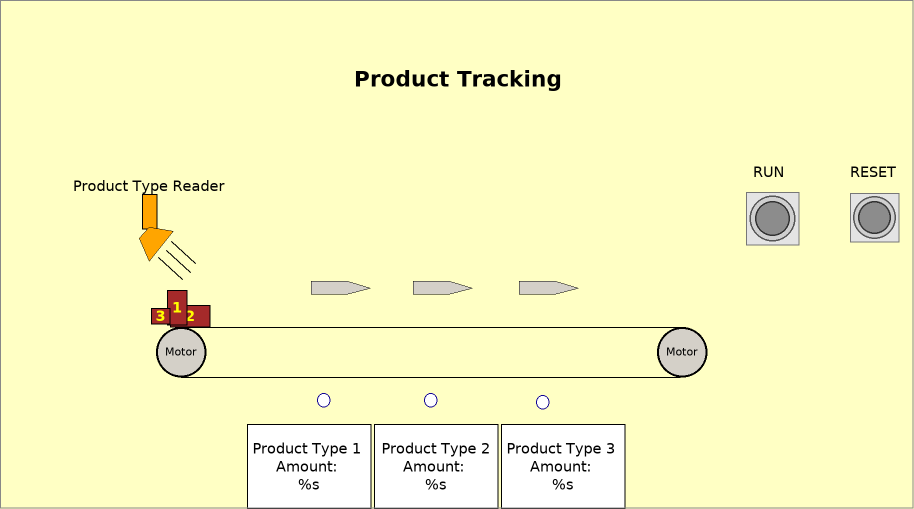
VISUALIZATION Visualization  // 914x509
    PushSwitchLed (746,191 53x55), variable: Simulation.CmdDrv01, behaviour: TOGGLE, style: Switch-PushSwitchLed-Gray
    Ellipse (156,327 50x50), "Motor", colour toggle: Simulation.Drive01.DrvRunning
    Label (728,157 82x30), "RUN"
    Label (832,157 82x30), "RESET"
    Ellipse (657,327 50x50), "Motor", colour toggle: Simulation.Drive01.DrvRunning
    Line (183,327) (680,327)
    Rectangle (142,194 15x35), angle 310
    Label (64,171 170x30), "Product Type Reader"
    Line (181,377) (680,377)
    Polygon (311,281) (347,281) (370,288) (347,294) (311,294)
        p2858320360: BOOL_TO_INT(MAIN.ConveyorTracking01.DiverterCmd) * 90
    Polygon (413,281) (449,281) (472,288) (449,294) (413,294)
        p2858320360: BOOL_TO_INT(MAIN.ConveyorTracking02.DiverterCmd) * 90
    Polygon (519,281) (555,281) (578,288) (555,294) (519,294)
        p2858320360: BOOL_TO_INT(MAIN.ConveyorTracking03.DiverterCmd) * 90
    Rectangle (170,305 40x22), "2", invisible if: Simulation.ProductType <> 2 OR MAIN.ConveyorTracking02.DistanceMoved > 52
        p3560616238: MAIN.ConveyorTracking02.DistanceMoved * 3.9
    Rectangle (167,290 20x35), "1", invisible if: Simulation.ProductType <> 1 OR MAIN.ConveyorTracking01.DistanceMoved > 32
        p3560616238: MAIN.ConveyorTracking01.DistanceMoved * 4.0
    Rectangle (151,308 19x16), "3", invisible if: Simulation.ProductType <> 3 OR MAIN.ConveyorTracking03.DistanceMoved > 72
        p3560616238: MAIN.ConveyorTracking03.DistanceMoved * 4.8
    Rectangle (247,424 124x85), "Product Type 1 Amount: %s", text variable: MAIN.DroppedProducts1.CV
    Ellipse (317,393 13x14), colour toggle: Simulation.tonProdType1Dropped.Q
    Ellipse (424,393 13x14), colour toggle: Simulation.tonProdType2Dropped.Q
    Ellipse (536,395 13x14), colour toggle: Simulation.tonProdType3Dropped.Q
    PushSwitch (850,191 49x53), variable: MAIN.Reset, behaviour: TAP, style: Switch-PushSwitch-Gray
    Rectangle (374,424 124x85), "Product Type 2 Amount: %s", text variable: MAIN.DroppedProducts2.CV
    Rectangle (501,424 124x85), "Product Type 3 Amount: %s", text variable: MAIN.DroppedProducts3.CV
    Label (322,64 272x30), "Product Tracking"
    Polygon (139,238) (149,227) (173,231) (149,261), colour toggle: Simulation.tpProductTypeRead.Q
    Line (171,241) (195,263), invisible if: NOT Simulation.tpProductTypeRead.Q
        p2086823670: NOT Simulation.tpProductTypeRead.Q
    Line (166,250) (190,272), invisible if: NOT Simulation.tpProductTypeRead.Q
        p2086823670: NOT Simulation.tpProductTypeRead.Q
    Line (158,257) (182,279), invisible if: NOT Simulation.tpProductTypeRead.Q
        p2086823670: NOT Simulation.tpProductTypeRead.Q
END_VISUALIZATION

(* stored: Version 1.1.0.1, ProductVersion 3.1.4024.15
   Visu Visualization: Id {69d51047-4eea-488d-8145-05668e8b9574} *)
